FUNCTION_BLOCK CAN_Object_Testing
VAR_INPUT
	NodeID			: BYTE; (* This Port No. addresses the CANopen Node (see System Manager) *)
	Start			: BOOL;
END_VAR
VAR_OUTPUT
	Finished		: BOOL;
END_VAR
VAR_IN_OUT
	CAN_Objects		: ARRAY [*] OF ST_CAN_Object;
END_VAR
VAR
	State			: BYTE := 0;
	Index			: DINT := 0;
	i				: BYTE := 0;
	
	Data		: ARRAY [0..255] OF BYTE;
	
	NMT_WRITE		: FB_NMT_WRITE;
	SDO_READ		: FB_SDO_READ;
	SDO_WRITE		: FB_SDO_WRITE;	
			
	RPDO_Nr				: BYTE := 3;	
	RPDO_Current_Number	: BYTE := 0;
	RPDO_Current_Mapped	: DWORD := 0;	
	
	TPDO_Nr				: BYTE := 3;
	TPDO_Current_Number	: BYTE := 0;
	TPDO_Current_Mapped	: DWORD := 0;
END_VAR

IF Start AND State = 255 THEN 
	State := 0;
END_IF

SDO_READ(StartReading:=FALSE);
SDO_WRITE(StartWriting:=FALSE);
NMT_WRITE(StartWriting:=FALSE);


CASE State OF	
	// ********** Initial steps **********	
	0: // NMT Set to Preoperational
		IF Start THEN
			NMT_WRITE(
				AdsNetID	:= GLB.ADSNetID_CAN,
				PortNr		:= 16#1000 + GLB.NodeID,
				ADSSTATE	:= ADSSTATE_RUN, 
				DEVSTATE	:= 0,
				StartWriting:=TRUE			
			);	
			State := State + 1;			
		END_IF
		
	1: // Wait for finish			
			IF NMT_WRITE.WriteDataFinished THEN
				Index := 0;	
				State := State + 1;	
			END_IF

			
	2:	// RPDO disable
		Data[3] := 16#80;
		Data[2] := 0;			
		Data[1] := RPDO_Nr + 1;
		Data[0] := NodeID;	
			
		SDO_WRITE(
			ADSNetID		:= GLB.ADSNetID_CAN,
			PortNr 		 	:= 16#1000 + GLB.NodeID,
			CO_Index 	 	:= 16#1400 + RPDO_Nr,
			CO_SubIndex  	:= 1,
			DataLength 	 	:= 4,
			StartWriting 	:= TRUE,
			WriteData 	 	:= Data );
		State := State + 1;	
		
	3: // Wait for finish
		IF SDO_WRITE.WriteDataFinished THEN
			State := State + 1;
		END_IF	
		
		
	4:	// RPDO Current Number of mapped objects
		SDO_READ(
			ADSNetID		:= GLB.ADSNetID_CAN,				
			PortNr 		 	:= 16#1000 + GLB.NodeID,
			CO_Index 		:= 16#1600 + RPDO_Nr,
			CO_SubIndex 	:= 0,
			DataLength 		:= 1,
			StartReading	:= TRUE	);
		State := State + 1;	
		
	5: // Wait for finish
		IF SDO_READ.ReadDataAvailable THEN
			RPDO_Current_Number := SDO_READ.ReadData[0];
			State := State + 1;
		END_IF
		
	
	6:	// RPDO Current mapped object
		SDO_READ(
			ADSNetID		:= GLB.ADSNetID_CAN,				
			PortNr 		 	:= 16#1000 + GLB.NodeID,
			CO_Index 		:= 16#1600 + RPDO_Nr,
			CO_SubIndex 	:= 1,
			DataLength 		:= 4,
			StartReading	:= TRUE);
		State := State + 1;	
		
	7: // Wait for finish
		IF SDO_READ.ReadDataAvailable THEN
			RPDO_Current_Mapped := SHL(BYTE_TO_DWORD(SDO_READ.ReadData[3]),24) + SHL(BYTE_TO_DWORD(SDO_READ.ReadData[2]),16) + SHL(BYTE_TO_DWORD(SDO_READ.ReadData[1]),8) + BYTE_TO_DWORD(SDO_READ.ReadData[0]);								
			State := State + 1;
		END_IF		
			
		
	8:	// TPDO disable
		Data[3] := 16#80;
		Data[2] := 0;			
		Data[1] := TPDO_Nr;
		Data[0] := NodeID + 16#80;	
			
		SDO_WRITE(
			ADSNetID		:= GLB.ADSNetID_CAN,
			PortNr 		 	:= 16#1000 + GLB.NodeID,
			CO_Index 	 	:= 16#1800 + TPDO_Nr,
			CO_SubIndex  	:= 1,
			DataLength 	 	:= 4,
			StartWriting 	:= TRUE,
			WriteData 	 	:= Data );		
		State := State + 1;	
		
	9: // Wait for finish
		IF SDO_WRITE.WriteDataFinished THEN
			State := State + 1;
		END_IF	
		

	10:	// TPDO Current Number of mapped objects
		SDO_READ(
			ADSNetID		:= GLB.ADSNetID_CAN,				
			PortNr 		 	:= 16#1000 + GLB.NodeID,
			CO_Index 		:= 16#1A00 + TPDO_Nr,
			CO_SubIndex 	:= 0,
			DataLength 		:= 1,
			StartReading	:= TRUE	);		
		State := State + 1;	
		
	11: // Wait for finish
		IF SDO_READ.ReadDataAvailable THEN
			TPDO_Current_Number := SDO_READ.ReadData[0];			
			State := State + 1;
		END_IF
		

	12:	// TPDO Current mapped object
		SDO_READ(
			ADSNetID		:= GLB.ADSNetID_CAN,				
			PortNr 		 	:= 16#1000 + GLB.NodeID,
			CO_Index 		:= 16#1A00 + TPDO_Nr,
			CO_SubIndex 	:= 1,
			DataLength 		:= 4,
			StartReading	:= TRUE	);		
		State := State + 1;	
		
	13: // Wait for finish
		IF SDO_READ.ReadDataAvailable THEN
			TPDO_Current_Mapped := SHL(BYTE_TO_DWORD(SDO_READ.ReadData[3]),24) + SHL(BYTE_TO_DWORD(SDO_READ.ReadData[2]),16) + SHL(BYTE_TO_DWORD(SDO_READ.ReadData[1]),8) + BYTE_TO_DWORD(SDO_READ.ReadData[0]);							
			State := 16;
		END_IF		
		
		
		
	// ********** Test steps **********
	16:	// Init
		IF CAN_Objects[Index].Length_Tested THEN 
			CAN_Objects[Index].Length_Tested := FALSE;
			CAN_Objects[Index].Length_Error := 0;
		ELSE
			CAN_Objects[Index].Length_Target := CAN_Objects[Index].Length; 
		END_IF
		
		IF CAN_Objects[Index].Readable_Tested THEN 
			CAN_Objects[Index].Readable_Tested := FALSE;
			CAN_Objects[Index].Readable_Error := 0;
			CAN_Objects[Index].Read_Value := 0;
		ELSE
			CAN_Objects[Index].Readable_Target := CAN_Objects[Index].Readable;
		END_IF
		
		IF CAN_Objects[Index].Writable_Tested THEN 
	    	CAN_Objects[Index].Writable_Tested := FALSE;
			CAN_Objects[Index].Writable_Error := 0; 
			CAN_Objects[Index].Write_Value := 0;
		ELSE		
			CAN_Objects[Index].Writable_Target := CAN_Objects[Index].Writable;
		END_IF
				
		IF CAN_Objects[Index].RPDO_Mappable_Tested THEN 
	    	CAN_Objects[Index].RPDO_Mappable_Tested := FALSE;
			CAN_Objects[Index].RPDO_Mappable_Error := 0; 
		ELSE		
			CAN_Objects[Index].RPDO_Mappable_Target := CAN_Objects[Index].RPDO_Mappable;
		END_IF
		
		IF CAN_Objects[Index].TPDO_Mappable_Tested THEN 
	    	CAN_Objects[Index].TPDO_Mappable_Tested := FALSE;
			CAN_Objects[Index].TPDO_Mappable_Error := 0; 
		ELSE		
			CAN_Objects[Index].TPDO_Mappable_Target := CAN_Objects[Index].TPDO_Mappable;
		END_IF	

		State := State + 1;
			
		
	17:	// Read Test
		SDO_READ(
			ADSNetID		:= GLB.ADSNetID_CAN,				
			PortNr 		 	:= 16#1000 + GLB.NodeID,
			CO_Index 		:= CAN_Objects[Index].Index,
			CO_SubIndex 	:= CAN_Objects[Index].Subindex,
			DataLength 		:= CAN_Objects[Index].Length,
			StartReading	:= TRUE	);		
		State := State + 1;
		
	18: // Read Test, wait for finish
		IF SDO_READ.ReadDataAvailable THEN
			CAN_Objects[Index].Readable_Tested := TRUE;
			CAN_Objects[Index].Read_Value := SHL(BYTE_TO_DWORD(SDO_READ.ReadData[3]),24) + SHL(BYTE_TO_DWORD(SDO_READ.ReadData[2]),16) + SHL(BYTE_TO_DWORD(SDO_READ.ReadData[1]),8) + BYTE_TO_DWORD(SDO_READ.ReadData[0]);	
			CAN_Objects[Index].Readable_Error := SDO_READ.Error;
			
			// LENGTH setzen !!!	
								
			State := State + 1;
		END_IF
	
		
	19:	// Write Test
		IF CAN_Objects[Index].Write_Value_Usage THEN CAN_Objects[Index].Write_Value := CAN_Objects[Index].Read_Value; END_IF
		FOR i := 0 TO CAN_Objects[Index].Length - 1 DO
			Data[i] := DWORD_TO_BYTE(SHR(CAN_Objects[Index].Write_Value, (8*i)));
		END_FOR;
			
		SDO_WRITE(
			ADSNetID	:= GLB.ADSNetID_CAN,
			PortNr 		 := 16#1000 + GLB.NodeID,
			CO_Index 	 := CAN_Objects[Index].Index,
			CO_SubIndex  := CAN_Objects[Index].Subindex,
			DataLength 	 := CAN_Objects[Index].Length,
			StartWriting := TRUE,
			WriteData 	 := Data );		
		State := State + 1;
			
	20: // Write Test, wait for finish
		IF SDO_WRITE.WriteDataFinished THEN
			CAN_Objects[Index].Writable_Tested := TRUE;
			CAN_Objects[Index].Write_Value := SHL(BYTE_TO_DWORD(SDO_Write.WriteData[3]),24) + SHL(BYTE_TO_DWORD(SDO_Write.WriteData[2]),16) + SHL(BYTE_TO_DWORD(SDO_Write.WriteData[1]),8) + BYTE_TO_DWORD(SDO_Write.WriteData[0]);				
			CAN_Objects[Index].Writable_Error := SDO_WRITE.Error;
			
			
			// Falls Read-Test nicht erfolgreich -> LENGTH hier setzen !!!	
			
		
			State := State + 1;
		END_IF

		
	21: // RPDO test	
		Data[0] := CAN_Objects[Index].Length * 8;
		Data[1] := CAN_Objects[Index].SubIndex;
		Data[2] := DWORD_TO_BYTE(CAN_Objects[Index].Index);
		Data[3] := DWORD_TO_BYTE(SHR(CAN_Objects[Index].Index,8));
			
		SDO_WRITE(
			ADSNetID	:= GLB.ADSNetID_CAN,
			PortNr 		 := 16#1000 + GLB.NodeID,
			CO_Index 	 := 16#1600 + RPDO_Nr,
			CO_SubIndex  := 1,
			DataLength 	 := 4,
			StartWriting := TRUE,
			WriteData 	 := Data );	
		State := State + 1;
			
	22: // RPDO test, wait for finish
		IF SDO_WRITE.WriteDataFinished THEN
			CAN_Objects[Index].RPDO_Mappable_Tested := TRUE;
			CAN_Objects[Index].RPDO_Mappable_Error := SDO_WRITE.Error;
									
			State := State + 1;
		END_IF	

				
	23: // TPDO test
		// Value for TPDO test is the same like RPDO test
 
		SDO_WRITE(
			ADSNetID	:= GLB.ADSNetID_CAN,
			PortNr 		 := 16#1000 + GLB.NodeID,
			CO_Index 	 := 16#1A00 + TPDO_Nr,
			CO_SubIndex  := 1,
			DataLength 	 := 4,
			StartWriting := TRUE,
			WriteData 	 := Data );	
		State := State + 1;
			
	24: // TPDO test, wait for finish
		IF SDO_WRITE.WriteDataFinished THEN
			CAN_Objects[Index].TPDO_Mappable_Tested := TRUE;
			CAN_Objects[Index].TPDO_Mappable_Error := SDO_WRITE.Error;
			
			State := State + 1;
		END_IF
		
		
	25: // Next object
		CAN_Objects[Index].Error := (CAN_Objects[Index].Readable_Error > 0) OR (CAN_Objects[Index].Writable_Error > 0) OR (CAN_Objects[Index].RPDO_Mappable_Error > 0) OR (CAN_Objects[Index].TPDO_Mappable_Error > 0);
			
		IF Index < UPPER_BOUND(CAN_Objects,1) THEN
			Index := Index + 1;
			State := 16;
		ELSE
			State := 128;
		END_IF
	
		
	// ********** Ending steps **********		
	128: // RPDO Reset mapped object
		Data[0] := DWORD_TO_BYTE(RPDO_Current_Mapped);
		Data[1] := DWORD_TO_BYTE(SHR(RPDO_Current_Mapped,8));
		Data[2] := DWORD_TO_BYTE(SHR(RPDO_Current_Mapped,16));
		Data[3] := DWORD_TO_BYTE(SHR(RPDO_Current_Mapped,24));
		SDO_WRITE(
			ADSNetID		:= GLB.ADSNetID_CAN,			
			PortNr 		 	:= 16#1000 + GLB.NodeID,
			CO_Index 		:= 16#1600 + TPDO_Nr,
			CO_SubIndex 	:= 1,
			DataLength 		:= 4,
			StartWriting	:= TRUE,
			WriteData 	 	:= Data );
		State := State + 1;
			
	129: // RPDO Reset mapped object, wait for finish		
		IF SDO_WRITE.WriteDataFinished THEN
			State := State + 1;
		END_IF		
			
		
	130: // RPDO Reset Number of mapped objects
		Data[0] := RPDO_Current_Number;
			
		SDO_WRITE(
			ADSNetID		:= GLB.ADSNetID_CAN,
			PortNr 		 	:= 16#1000 + GLB.NodeID,
			CO_Index 		:= 16#1600 + RPDO_Nr,
			CO_SubIndex 	:= 0,
			DataLength 		:= 1,
			StartWriting 	:= TRUE,
			WriteData 	 	:= Data );
		State := State + 1;
			
	131: // RPDO Reset Number of mapped objects, wait for finish			
		IF SDO_WRITE.WriteDataFinished THEN
			State := State + 1;
		END_IF			

		
	132: // RPDO reactivate
		Data[3] := 0;
		Data[2] := 0;			
		Data[1] := RPDO_Nr + 1;
		Data[0] := NodeID;	
			
		SDO_WRITE(
			ADSNetID	:= GLB.ADSNetID_CAN,
			PortNr 		 := 16#1000 + GLB.NodeID,
			CO_Index 	 := 16#1400 + RPDO_Nr,
			CO_SubIndex  := 1,
			DataLength 	 := 4,
			StartWriting := TRUE,
			WriteData 	 := Data );
		State := State + 1;
			
	133: // RPDO reactivate, wait for finish	
		IF SDO_WRITE.WriteDataFinished THEN
			State := State + 1;
		END_IF	
		
		
	134: // TPDO Reset mapped object
		Data[0] := DWORD_TO_BYTE(TPDO_Current_Mapped);
		Data[1] := DWORD_TO_BYTE(SHR(TPDO_Current_Mapped,8));
		Data[2] := DWORD_TO_BYTE(SHR(TPDO_Current_Mapped,16));
		Data[3] := DWORD_TO_BYTE(SHR(TPDO_Current_Mapped,24));
		
		SDO_WRITE(
			ADSNetID		:= GLB.ADSNetID_CAN,			
			PortNr 		 	:= 16#1000 + GLB.NodeID,
			CO_Index 		:= 16#1A00 + TPDO_Nr,
			CO_SubIndex 	:= 1,
			DataLength 		:= 4,
			StartWriting	:= TRUE,
			WriteData 	 	:= Data );
		State := State + 1;
			
	135: // TPDO Reset mapped object, wait for finish	
		IF SDO_WRITE.WriteDataFinished THEN
			State := State + 1;
		END_IF			
			
		
	136:// TPDO Reset Number of mapped objects
		Data[0] := TPDO_Current_Number;
			
		SDO_WRITE(
			ADSNetID		:= GLB.ADSNetID_CAN,
			PortNr 		 	:= 16#1000 + GLB.NodeID,
			CO_Index 		:= 16#1A00 + RPDO_Nr,
			CO_SubIndex 	:= 0,
			DataLength 		:= 1,
			StartWriting 	:= TRUE,
			WriteData 	 	:= Data );
		State := State + 1;
			
	137: // TPDO Reset Number of mapped objects, wait for finish	
		IF SDO_WRITE.WriteDataFinished THEN
			State := State + 1;
		END_IF			

		
	138: // TPDO reactivate
		Data[3] := 0;
		Data[2] := 0;			
		Data[1] := TPDO_Nr;
		Data[0] := NodeID + 16#80;	
			
		SDO_WRITE(
			ADSNetID	:= GLB.ADSNetID_CAN,
			PortNr 		 := 16#1000 + GLB.NodeID,
			CO_Index 	 := 16#1400 + RPDO_Nr,
			CO_SubIndex  := 1,
			DataLength 	 := 4,
			StartWriting := TRUE,
			WriteData 	 := Data );
		State := State + 1;
			
	139: // TPDO reactivate, wait for finish	
		IF SDO_WRITE.WriteDataFinished THEN
			State := State + 1;
		END_IF	
						
	
	140: // NMT Set to operational
		NMT_WRITE(
			ADSNetID	:= GLB.ADSNetID_CAN,
			PORTNr		:= 16#1000 + GLB.NodeID,
			ADSSTATE	:= ADSSTATE_RUN,
			DEVSTATE	:= 1,
			StartWriting:=TRUE );	
		State := State + 1;
			
	141: // RPDO Reset Number of mapped objects, wait for finish	
		IF NMT_WRITE.WriteDataFinished THEN
			State := 255;	
		END_IF

		
	// ********** End **********
	ELSE	// Tests finished	
		Finished := TRUE;
		State := 255;
			
END_CASE

END_FUNCTION_BLOCK

(* stored: Version 1.1.0.1, ProductVersion 3.1.4024.11
   POU CAN_Object_Testing: Id {90e6a8ef-3c73-461e-85bb-0bda0ca2917c}, SpecialFunc None *)
